(* CoDeSys 2.3.9.37 project: Gemma.pro *)
(* Libraries: Standard.lib 4.10.05 12:14:46, IecSfc.lib 13.4.06 16:51:28 *)

(* Global variable list: Global_Variables *)
VAR_GLOBAL

(* Variables de Entrada *)
   A1:BOOL;
   A2:BOOL;
   B1:BOOL;
   B2:BOOL;
   SensorPieza:BOOL;
   PiezaEnSistema:BOOL;
   MANUAL:BOOL;  (*  Modo MANUAL/AUTOMATICO *)
   EMERGENCIA:BOOL;  (* Seta de Emergencia *)
   CONEXION:BOOL;  (* Interruptor de conexion *)
   M:BOOL;
   P:BOOL;
   Rearme:BOOL;
   BotonExt1:BOOL;
   BotonRet1:BOOL;
   BotonExt2:BOOL;
   BotonRet2:BOOL;


(* Variables de Salida *)
   Cil1Ext:BOOL;
   Cil1Ret:BOOL;
   Cil2Ext:BOOL;
   Cil2Ret:BOOL;
   LuzEmergencia:BOOL;
   EnServicio:BOOL;
   EnOperacionAuto:BOOL;
   EnOperacionManual:BOOL;


END_VAR

(* POU PLC_PRG, ST *)
PROGRAM PLC_PRG
VAR
END_VAR
Proceso();
END_PROGRAM

(* POU Proceso, ST *)
PROGRAM Proceso
VAR
	posy1: INT;
	posPiezay:INT :=1000;
	posy2: INT;
	posPiezax:INT := 1000;
	PonPieza: BOOL;
       QuitaPieza:BOOL;
END_VAR
IF Cil1Ext=TRUE AND posy1<100 THEN
 IF posPiezay=posy1 AND posPiezax<36 THEN
          posPiezay:=posPiezay+1;
   END_IF
   posy1:=posy1+1;
END_IF

IF Cil1Ret=TRUE AND posy1>0 THEN
    posy1:=posy1-3;
END_IF

IF posy1<=0 THEN
  A1:=TRUE;
ELSE
  A1:=FALSE;
END_IF

IF posy1>=100 THEN
  A2:=TRUE;
ELSE
  A2:=FALSE;
END_IF


IF Cil2Ext=TRUE AND posy2<120  THEN
 IF posPiezax+20=posy2 AND posPiezay>65 THEN
          posPiezax:=posPiezax+1;
   END_IF
   posy2:=posy2+1;
END_IF

IF Cil2Ret=TRUE AND posy2>0 THEN
    posy2:=posy2-3;
END_IF

IF posy2<=0 THEN
  B1:=TRUE;
ELSE
  B1:=FALSE;
END_IF

IF posy2>=120 THEN
  B2:=TRUE;
ELSE
  B2:=FALSE;
END_IF

IF posPiezay=1000 AND posPiezax=1000 AND PonPieza THEN
    posPiezax:=0;
   posPiezay:=0;
END_IF

IF QuitaPieza THEN
	posPiezay:=1000;
       posPiezax:=1000;
END_IF

IF posPiezax=100 THEN
    posPiezax:=1000;
   posPiezay:=1000;
END_IF

IF PosPiezay<28 THEN
   SensorPieza:=TRUE;
ELSE
   SensorPieza:=FALSE;
END_IF


IF PosPiezay<200 AND PosPiezay<200 THEN
   PiezaEnSistema:=TRUE;
ELSE
   PiezaEnSistema:=FALSE;
END_IF
END_PROGRAM

(* Visualisation CuadroControl
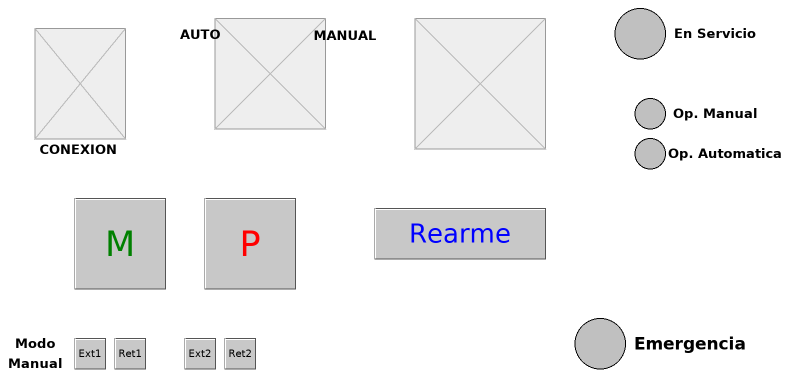
bitmap at (220,50)-(331,161): SELECTOR1.BMP
bitmap at (220,50)-(331,161): SELECTOR2.BMP
rectangle at (310,52)-(391,83): text "MANUAL"
rectangle at (165,51)-(246,82): text "AUTO"
bitmap at (420,50)-(551,181): EMERGENCIA1.BMP
bitmap at (420,50)-(551,181): EMERGENCIA2.BMP
button at (80,230)-(171,321): text "M"; taps M
button at (210,230)-(301,321): text "P"; taps P
button at (380,240)-(551,291): text "Rearme"; taps Rearme
bitmap at (40,60)-(131,171): ON.BMP
bitmap at (40,60)-(131,171): OFF.BMP
ellipse at (620,40)-(671,91): alarm colour if EnServicio
rectangle at (680,50)-(761,81): text "En Servicio"
ellipse at (640,130)-(671,161): alarm colour if EnOperacionManual
rectangle at (680,130)-(761,161): text "Op. Manual"
ellipse at (640,170)-(671,201): alarm colour if EnOperacionAuto
rectangle at (670,170)-(791,201): text "Op. Automatica"
ellipse at (580,350)-(631,401): alarm colour if LuzEmergencia
rectangle at (630,360)-(761,391): text "Emergencia"
button at (80,370)-(111,401): text "Ext1"; toggles BotonExt1
button at (120,370)-(151,401): text "Ret1"; toggles BotonRet1
rectangle at (0,360)-(81,391): text "Modo"
rectangle at (0,380)-(81,411): text "Manual"
button at (190,370)-(221,401): text "Ext2"; toggles BotonExt2
button at (230,370)-(261,401): text "Ret2"; toggles BotonRet2
rectangle at (43,166)-(124,197): text "CONEXION"
*)

(* Visualisation Proceso
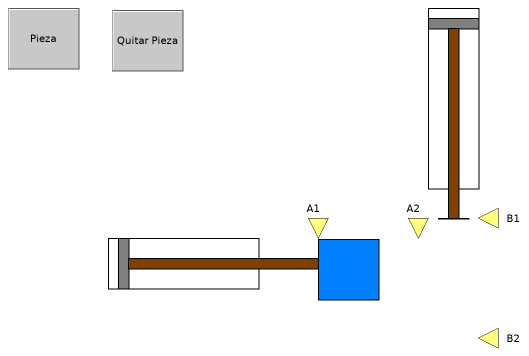
rectangle at (330,320)-(431,361): text "SensorPieza"
polygon at (340,270)-(360,290): alarm colour if A1; toggles .B
rectangle at (150,290)-(161,341): left Proceso.posy1; right Proceso.posy1
rectangle at (160,310)-(351,321): left Proceso.posy1; right Proceso.posy1
polygon at (440,270)-(460,290): alarm colour if A2; toggles .B
rectangle at (350,300)-(351,331): left Proceso.posy1; right Proceso.posy1
rectangle at (320,240)-(371,281): text "A1"
rectangle at (420,240)-(471,281): text "A2"
rectangle at (460,60)-(511,241): angle 90
rectangle at (460,70)-(511,81): top Proceso.posy2; bottom Proceso.posy2
rectangle at (480,80)-(491,271): top Proceso.posy2; bottom Proceso.posy2
rectangle at (520,250)-(571,291): text "B1"
rectangle at (520,370)-(571,411): text "B2"
polygon at (510,260)-(530,280): alarm colour if B1
rectangle at (350,291)-(411,352): left Proceso.posPiezay; top Proceso.posPiezax; right Proceso.posPiezay; bottom Proceso.posPiezax
polygon at (510,380)-(530,400): alarm colour if B2
rectangle at (470,270)-(501,271): top Proceso.posy2; bottom Proceso.posy2
button at (40,60)-(111,121): text "Pieza"; taps Proceso.PonPieza
button at (144,62)-(215,123): text "Quitar Pieza"; taps Proceso.QuitaPieza
2 more shapes without text or variables
*)
